FUNCTION_BLOCK FB_SUB_INT (* INT Subtraction *)
  (* Standard: 61499-1-D.1; Classification: Math *)
  (* Version 0.0, 2002-03-13, JHC, Rockwell Automation *)
  (* Compiler header: package fb.rt.math; *)
  (* Compiler classdef: class FB_SUB_DINT extends FB_ADD_INT *)
  (* Compiler Java IBM VisualAge 3.0 *)
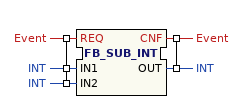
  EVENT_INPUT
    REQ WITH IN1, IN2;
  END_EVENT
  EVENT_OUTPUT
    CNF WITH OUT;
  END_EVENT
  VAR_INPUT
    IN1 : INT; (* Minuend *)
    IN2 : INT; (* Subtrahend *)
  END_VAR
  VAR_OUTPUT
    OUT : INT; (* Difference *)
  END_VAR
END_FUNCTION_BLOCK
